FUNCTION_BLOCK eigvec_in (* Basic FB with empty ECC *)
  (* Standard: 61499-2 *)
  (* Version 1.0, 2020-08-21, Administrator *)
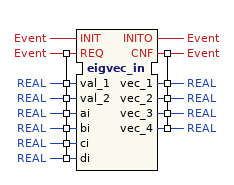
  EVENT_INPUT
    INIT;
    REQ WITH val_1, val_2, ai, bi, ci, di;
  END_EVENT
  EVENT_OUTPUT
    INITO;
    CNF WITH vec_1, vec_2, vec_3, vec_4;
  END_EVENT
  VAR_INPUT
    val_1 : REAL;
    val_2 : REAL;
    ai : REAL;
    bi : REAL;
    ci : REAL;
    di : REAL;
  END_VAR
  VAR_OUTPUT
    vec_1 : REAL;
    vec_2 : REAL;
    vec_3 : REAL;
    vec_4 : REAL;
  END_VAR
  VAR
    x1 : REAL; (* Internal Variable *)
    x2 : REAL; (* Internal Variable *)
    y1 : REAL; (* Internal Variable *)
    y2 : REAL; (* Internal Variable *)
    divisor : REAL; (* Internal Variable *)
    x : REAL; (* Internal Variable *)
    y : REAL; (* Internal Variable *)
    x1_2 : REAL; (* Internal Variable *)
    x2_2 : REAL; (* Internal Variable *)
    m1 : REAL; (* Internal Variable *)
    m2 : REAL; (* Internal Variable *)
    m3 : REAL; (* Internal Variable *)
    m4 : REAL; (* Internal Variable *)
  END_VAR
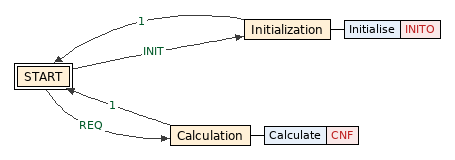
  EC_STATES
    START; (* Initial State *)
    Initialization : Initialise -> INITO;
    Calculation : Calculate -> CNF;
  END_STATES
  EC_TRANSITIONS
    Initialization TO START := 1;
    START TO Initialization := INIT;
    Calculation TO START := 1;
    START TO Calculation := REQ;
  END_TRANSITIONS
  ALGORITHM Initialise IN ST: (* New Algorithm *)

  END_ALGORITHM
  ALGORITHM Calculate IN ST: (* New Algorithm *)
x1 := ai-val_1;
x2 := bi;
y1 := ci;
y2 := di-val_2;

x1_2 := EXPT(x1,2);
x2_2 := EXPT(x2,2);

x := x1_2 + x2_2;

divisor := SQRT(x);

///

IF  (bi>0) and (di<0) and (ai>0) and ( ABS(di)>ai ) THEN //1
	m1 := -1;
	m2 := 1;
	m3 := -1;
	m4 := 1;
ELSIF (bi>0) and (di<0) and (ai<0) and (ABS(di)>ABS(ai)) THEN //2
	m1 := -1;
	m2 := 1;
	m3 := -1;
	m4 := 1;
ELSIF (bi>0) and (di>0) and (ai>0) and (di>ai) THEN //3
	m1 := -1;
	m2 := -1;
	m3 := -1;
	m4 := -1;
ELSIF (bi>0) and (di<0) and (ai<0) and (abs(di)=abs(ai)) THEN //4
	m1 := 1;
	m2 := -1;
	m3 := 1;
	m4 := -1;
ELSIF (bi>0) and (ai<0) and (di>0) and (ABS(ai)>di) THEN //5
	m1 := -1;
	m2 := 1;
	m3 := -1;
	m4 := 1;
ELSIF (bi<0) and (ai<0) and (di<0) and (ABS(di)>ABS(ai)) THEN //6
	m1 := -1;
	m2 := 1;
	m3 := -1;
	m4 := 1;
ELSIF (bi<0) and (ai<0) and (di<0) and (ABS(di)<ABS(ai)) THEN //7
	m1 := 1;
	m2 := -1;
	m3 := 1;
	m4 := -1;
ELSIF (bi<0) and (ai<0) and (di>0) and (ABS(di)<ABS(ai)) THEN //8
	m1 := 1;
	m2 := -1;
	m3 := 1;
	m4 := -1;
ELSIF (bi<0) and (ai<0) and (di<0) and (ABS(di)=ABS(ai)) THEN //9
	m1 := -1;
	m2 := 1;
	m3 := -1;
	m4 := 1;
ELSE
	m1 := 1;
	m2 := 1;
	m3 := 1;
	m4 := 1;
END_IF;

///

vec_1 := m1*x2/divisor;
vec_2 := m2*-x1/divisor;
vec_3 := m3*y2/divisor;
vec_4 := m4*-y1/divisor;
  END_ALGORITHM
END_FUNCTION_BLOCK
